FUNCTION TryConvert_UDINT_TO_UDINT : BOOL
VAR_INPUT
	in : UDINT;
	out : REFERENCE TO UDINT;
END_VAR

out := in;
TryConvert_UDINT_TO_UDINT := TRUE;

END_FUNCTION

(* stored: Version 1.1.0.1, ProductVersion 3.1.4024.12
   POU TryConvert_UDINT_TO_UDINT: Id {4ab931f1-5356-4712-b0c8-0bc9df2be179}, SpecialFunc None *)
